# EPICS autosave request: ADApp/Db/NDGatherN_settings.req
$(P)$(R)NDArrayPort_$(N)
$(P)$(R)NDArrayAddress_$(N)
